{attribute 'GeneratedUsingTerminal: EL2262-0000-0002'}
{attribute addProperty BoxType "EL2262-0000-0002"}
{attribute addProperty Id "Cycle_Counter0AT %Q*UINT2"}
{attribute addProperty CRC "2940411104"}
{attribute addProperty Size "2"}
TYPE CycCount0_AF431CE0 :
STRUCT
	{attribute addProperty Name "Cycle_Counter0"}
	Cycle_Counter0 AT %Q* : UINT;
END_STRUCT
END_TYPE

(* stored: Version 1.2.0.0, ProductVersion 3.1.4024.9
   DUT CycCount0_AF431CE0: Id {f875d2c5-d111-4413-9793-5872086d7722} *)
